{attribute addProperty BoxType "EL1258-0000-0016"}
{attribute addProperty Id "Input_event_state_1BIT10.12533Input_event_state_2BIT10.12534Input_event_state_3BIT10.12535Input_event_state_4BIT10.12536Input_event_state_5BIT10.12537Input_event_state_6BIT10.12538Input_event_state_7BIT10.12539Input_event_state_8BIT10.12540Input_event_state_9BIT10.12541Input_event_state_10BIT10.12542"}
{attribute addProperty CRC "2340108288"}
{attribute addProperty SizeInBites "186"}
{attribute addProperty SizeInBytes "23.25"}
{warning 'Size of this structure is not a multiple of 8 bits!!!'}
TYPE Inputs_8B7B3800 :
STRUCT
	{attribute addProperty Name "Input_event_state_1"}
	Input_event_state_1 : BIT;
	{attribute addProperty Name "Input_event_state_2"}
	Input_event_state_2 : BIT;
	{attribute addProperty Name "Input_event_state_3"}
	Input_event_state_3 : BIT;
	{attribute addProperty Name "Input_event_state_4"}
	Input_event_state_4 : BIT;
	{attribute addProperty Name "Input_event_state_5"}
	Input_event_state_5 : BIT;
	{attribute addProperty Name "Input_event_state_6"}
	Input_event_state_6 : BIT;
	{attribute addProperty Name "Input_event_state_7"}
	Input_event_state_7 : BIT;
	{attribute addProperty Name "Input_event_state_8"}
	Input_event_state_8 : BIT;
	{attribute addProperty Name "Input_event_state_9"}
	Input_event_state_9 : BIT;
	{attribute addProperty Name "Input_event_state_10"}
	Input_event_state_10 : BIT;
	{attribute 'hide'}
	reserve_2_BOOL_0 : BOOL;
	{attribute 'hide'}
	reserve_2_BOOL_1 : BOOL;
	{attribute 'hide'}
	reserve_2_BOOL_2 : BOOL;
	{attribute 'hide'}
	reserve_2_BOOL_3 : BOOL;
	{attribute 'hide'}
	reserve_2_BOOL_4 : BOOL;
	{attribute 'hide'}
	reserve_2_BOOL_5 : BOOL;
	{attribute 'hide'}
	reserve_2_BOOL_6 : BOOL;
	{attribute 'hide'}
	reserve_2_BOOL_7 : BOOL;
	{attribute 'hide'}
	reserve_2_BOOL_8 : BOOL;
	{attribute 'hide'}
	reserve_2_BOOL_9 : BOOL;
	{attribute 'hide'}
	reserve_2_BOOL_10 : BOOL;
	{attribute 'hide'}
	reserve_2_BOOL_11 : BOOL;
	{attribute 'hide'}
	reserve_2_BOOL_12 : BOOL;
	{attribute 'hide'}
	reserve_2_BOOL_13 : BOOL;
	{attribute 'hide'}
	reserve_2_BOOL_14 : BOOL;
	{attribute 'hide'}
	reserve_2_BOOL_15 : BOOL;
	{attribute 'hide'}
	reserve_2_BOOL_16 : BOOL;
	{attribute 'hide'}
	reserve_2_BOOL_17 : BOOL;
	{attribute 'hide'}
	reserve_2_BOOL_18 : BOOL;
	{attribute 'hide'}
	reserve_2_BOOL_19 : BOOL;
	{attribute 'hide'}
	reserve_2_BOOL_20 : BOOL;
	{attribute 'hide'}
	reserve_2_BOOL_21 : BOOL;
END_STRUCT
END_TYPE

(* stored: Version 1.2.0.0, ProductVersion 3.1.4024.9
   DUT Inputs_8B7B3800: Id {29d19358-5545-432f-97af-7159f7823e47} *)
